// TIA Portal V17 export
// export: Created 2024-09-02T12:50:16.4502207Z, ExportSetting WithDefaults, DisplayName Totally Integrated Automation Portal, DisplayVersion V17, DisplayName TIA Portal Openness, DisplayVersion V17, DisplayName TIA Portal Version Control Interface, DisplayVersion V17, DisplayName STEP 7 Professional, DisplayVersion V17, DisplayName STEP 7 Safety, DisplayVersion V17, DisplayName WinCC Professional, DisplayVersion V17
DATA_BLOCK "AnwDB_OperatingModes_OP70"   // DB61
{ S7_Optimized_Access := 'TRUE'; DB_Accessible_From_OPC_UA := 'FALSE' }
AUTHOR : OlegFuehrus
FAMILY : BA
NAME : BA
VERSION : 0.1
// stored: AutoNumber true, DBAccessibleFromOPCUA false, IsOnlyStoredInLoadMemory false, IsRetainMemResEnabled false, IsWriteProtectedInAS false, MemoryReserve 100
   VAR
      Global { S7_SetPoint := 'True'} : "TypeOperatingModesGlobal";
      BA { S7_SetPoint := 'True'} : Array[0..1] of "TypeOperatingModes";
      Central { ExternalWritable := 'False'} : Struct   // Einschaltung Zentrale / Switching on central
         Machine_On { ExternalWritable := 'False'} : Bool;   // Maschine einschalten / Switch on the machine
         Machine_Off { ExternalWritable := 'False'} : Bool;   // Maschine ausschalten / Switch off the machine
         HTE { ExternalWritable := 'False'} : Bool;   // Halt bei Taktende / Stop at end of cycle
         Start { ExternalWritable := 'False'} : Bool;   // Automatik starten / Start automatic
      END_STRUCT;
      Extern { ExternalWritable := 'False'} : Struct   // Einschaltung Extern / External switch-on
         Ready { ExternalWritable := 'False'} : Bool;   // Bereit fuer Externe einschaltung / Ready for external switch-on
         Auto { ExternalWritable := 'False'} : Bool;   // Anwahl BA Automatik / Selection BA Automatic
         Safety_Quit { ExternalWritable := 'False'} : Bool;   // Sicherheitskreise quittieren / Acknowledge safety circuits
         Medium_On { ExternalWritable := 'False'} : Bool;   // Medien einschalten / Switch on media
         Start_On { ExternalWritable := 'False'} : Bool;   // Start einschalten / Switch on start
         Error_Quit { ExternalWritable := 'False'} : Bool;   // Fehler quittieren / Acknowledge error
         Active { ExternalWritable := 'False'} : Bool;   // Externe Einschaltung aktiv / External switch-on active
      END_STRUCT;
      HMI : Struct
         Screen_active : Bool;
         BA_Choice : Int;
         BA { S7_SetPoint := 'True'} : Array[0..4] of "TypeOperatingModesHMI";
      END_STRUCT;
   END_VAR
BEGIN
   Global.machine_on := true;
END_DATA_BLOCK
